INTERFACE ITF_BaseComponent_HMI

END_INTERFACE

(* stored: Version 1.1.0.1
   Itf ITF_BaseComponent_HMI: Id {09893359-9aae-0055-210b-9fb2bfb82b06} *)
